Staubli VAL3: initvis.pgx

program initvis(bool& x_bResult[] (dimensions=1))
  local bool l_bResult
begin


  x_bResult=true
  clearBuffer(skVision)

end
